// TIA Portal project "2026_04_16_Progetto1" (V15)

(* hardware
DEVICE "S7-1200 station_1"  S7-1200 Station
   slot 0: "Telaio di montaggio_0"  S7-1200 Rack  Rack  V1.0
   slot 1: "PLC_1"  CPU 1215C DC/DC/DC  6ES7 215-1AG40-0XB0  V4.2
*)

// ===== PLC "PLC_1"  CPU 1215C DC/DC/DC =====

VAR_GLOBAL   // PLC tag table "Tabella delle variabili standard"
   "System_Byte" AT %MB1 : Byte;
   "FirstScan" AT %M1.0 : Bool;
   "DiagStatusUpdate" AT %M1.1 : Bool;
   "AlwaysTRUE" AT %M1.2 : Bool;
   "AlwaysFALSE" AT %M1.3 : Bool;
   "System_Byte(1)" AT %MB1 : Byte;
   "Clock_Byte" AT %MB0 : Byte;
   "Clock_10Hz" AT %M0.0 : Bool;
   "Clock_5Hz" AT %M0.1 : Bool;
   "Clock_2.5Hz" AT %M0.2 : Bool;
   "Clock_2Hz" AT %M0.3 : Bool;
   "Clock_1.25Hz" AT %M0.4 : Bool;
   "Clock_1Hz" AT %M0.5 : Bool;
   "Clock_0.625Hz" AT %M0.6 : Bool;
   "Clock_0.5Hz" AT %M0.7 : Bool;
   "P_start" AT %I2.0 : Bool;   // Pulsante di avvio
   "P_stop" AT %I2.1 : Bool;   // Pulsante di arresto
   "km" AT %Q0.0 : Bool;   // Contatto motore
   "KMA" AT %M100.0 : Bool;   // Stato enable motore
   "H" AT %Q0.1 : Bool;
END_VAR

// folder: System blocks/Program resources

DATA_BLOCK "IEC_Timer_0_DB"   // DB1
{ S7_Optimized_Access := 'TRUE' }
AUTHOR : Simatic
FAMILY : IEC
NAME : IEC_TMR
VERSION : 1.0
// stored: InstanceOfName IEC_TIMER
"IEC_TIMER"
BEGIN
END_DATA_BLOCK

// folder: (top level)

ORGANIZATION_BLOCK "Main"   // OB1, LAD, ProgramCycle
TITLE = "Main Program Sweep (Cycle)"
{ S7_Optimized_Access := 'TRUE' }
VERSION : 0.1
// Programma per gestire un motore
   VAR_INPUT
      Initial_Call : Bool;   // Initial call of this OB
      Remanence : Bool;   // =True, if remanent data are available
   END_VAR
BEGIN

REGION Network 1: Contatto motore
   // Gestione avvio motore (logica)
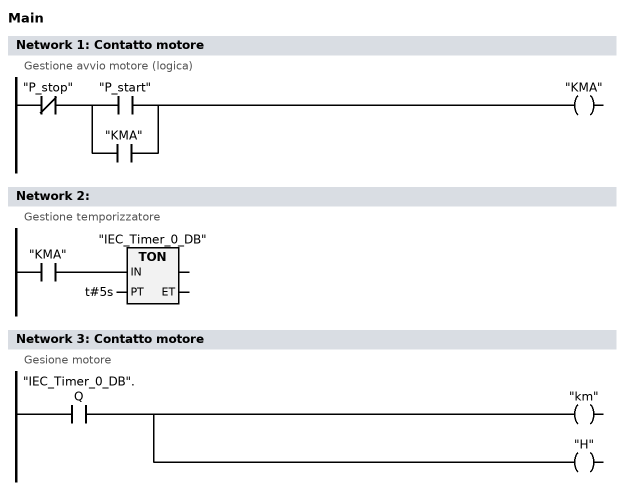
   RUNG wire#powerrail
      I_Contact( "P_stop" )
      wire#w1
      Contact( "P_start" )
      wire#w2
      Coil( "KMA" )
   END_RUNG
   RUNG wire#w1
      Contact( "KMA" )
   END_RUNG wire#w2
   // the same network as SCL:
   "KMA" := NOT "P_stop" AND ("P_start" OR "KMA");
END_REGION

REGION Network 2
   // Gestione temporizzatore
   "IEC_Timer_0_DB".TON(IN := "KMA", PT := t#5s);
END_REGION

REGION Network 3: Contatto motore
   // Gesione motore
   RUNG wire#powerrail
      Contact( "IEC_Timer_0_DB".Q )
      wire#w1
      Coil( "km" )
   END_RUNG
   RUNG wire#w1
      Coil( "H" )
   END_RUNG
   // the same network as SCL:
   "km" := "IEC_Timer_0_DB".Q;
   "H" := "IEC_Timer_0_DB".Q;
END_REGION
END_ORGANIZATION_BLOCK